KUKA KRL data list: AMM_Config.dat

&ACCESS RVO1
&REL 3
&PARAM EDITMASK = *
&PARAM TEMPLATE = C:\KRC\Roboter\Template\vorgabe
DEFDAT AMM_Config PUBLIC
;FOLD EXTERNAL DECLARATIONS;%{PE}%MKUKATPBASIS,%CEXT,%VCOMMON,%P
;FOLD BASISTECH EXT;%{PE}%MKUKATPBASIS,%CEXT,%VEXT,%P
EXT  BAS (BAS_COMMAND  :IN,REAL  :IN )
DECL INT SUCCESS
;ENDFOLD (BASISTECH EXT)
;FOLD USER EXT;%{E}%MKUKATPUSER,%CEXT,%VEXT,%P
;Make your modifications here


DECL GLOBAL INT gnMillFrequencyMax=4500  ; Max 22000
DECL GLOBAL INT gnMillFrequencyMin=10

DECL GLOBAL BOOL gbToolChangerPresent = true
DECL GLOBAL BOOL gbTCCoverPresent = FALSE
ENUM TYPAir MAINAIRON,MAINAIROFF,BLOWAIRON,BLOWAIROFF

;ENDFOLD (USER EXT)
;ENDFOLD (EXTERNAL DECLARATIONS)
ENDDAT
